// TIA Portal V16 export
// export: Created 2025-05-30T16:30:26.6325314Z, ExportSetting WithDefaults, DisplayName Totally Integrated Automation Portal, DisplayVersion V16, DisplayName TIA Portal Version Control Interface, DisplayVersion V16, DisplayName TIA Portal Openness, DisplayVersion V16, DisplayName STEP 7 Professional, DisplayVersion V16, DisplayName STEP 7 Safety, DisplayVersion V16, DisplayName WinCC Advanced, DisplayVersion V16
FUNCTION_BLOCK "MC_Move"   // FB10, FBD
TITLE = MC_Move
VERSION : 0.1
// Block moves an Axis to an Desired Position, this block comes with the brake feature. When the axis is on position it keeps the brake for a time. You can set the time in the Brake Time field.
// stored: AutoNumber true, IsIECCheckEnabled false, UDAEnableTagReadback false
   VAR_INPUT
      Start : Bool;
      "Desired Position" : Real;
      "Speed (50-75%)" : Int;
      "Brake on Position" : Bool;
      Acceleration : Real;
      Deacceleration : Real;
      "Drive Ready" : Bool;
      "Drive On Position" : Bool;
      "Brake Time" : Time := T#500ms;
      "Safety OK" : Bool;
   END_VAR
   VAR_OUTPUT
      Go : Bool;
      "Desired Position Out" : Real;
      "Speed Output" : Int;
      "Acceleration Out" : Real;
      "Deacceleration Out" : Real;
      "Brake Out" : Bool;
   END_VAR
   VAR_TEMP
      SR_1 : Bool;
   END_VAR
BEGIN

REGION Network 1: Start - Go To Position + Speed
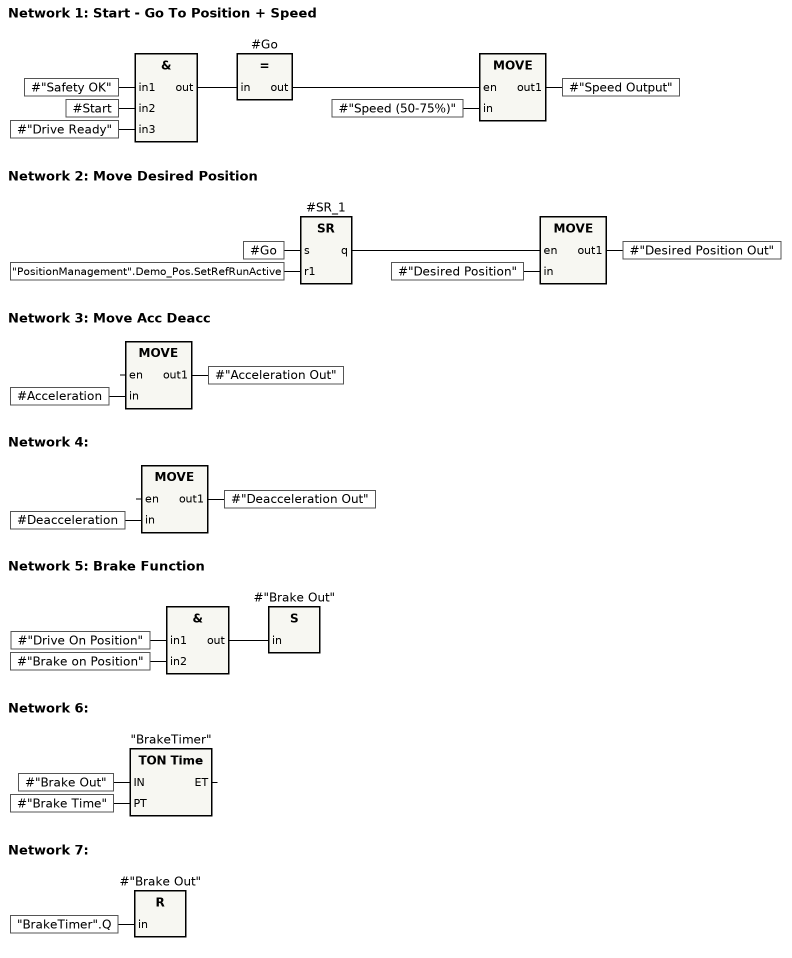
   #Go := #"Safety OK" AND #Start AND #"Drive Ready";
   IF #Go THEN #"Speed Output" := #"Speed (50-75%)"; END_IF;
END_REGION

REGION Network 2: Move Desired Position
   IF #Go THEN
       #SR_1 := TRUE;   // SR flip-flop
   END_IF;
   IF "PositionManagement".Demo_Pos.SetRefRunActive THEN #SR_1 := FALSE; END_IF;
   IF #SR_1 THEN #"Desired Position Out" := #"Desired Position"; END_IF;
END_REGION

REGION Network 3: Move Acc Deacc
   #"Acceleration Out" := #Acceleration;
END_REGION

REGION Network 4
   #"Deacceleration Out" := #Deacceleration;
END_REGION

REGION Network 5: Brake Function
   IF #"Drive On Position" AND #"Brake on Position" THEN #"Brake Out" := TRUE; END_IF;
END_REGION

REGION Network 6
   "BrakeTimer".TON(IN := #"Brake Out", PT := #"Brake Time");
END_REGION

REGION Network 7
   IF "BrakeTimer".Q THEN #"Brake Out" := FALSE; END_IF;
END_REGION
END_FUNCTION_BLOCK
